(* Logix 5000 project; controller CarbonScout_MK6 vendor 1 type 14 code 154 rev 32.11; software revision 32.00 *)
// CarbonScout_MK6

TASK DataMapping (periodic, rate 200 ms, priority 15, watchdog 1000 ms) : DataMapping
TASK Instruments (periodic, rate 100 ms, priority 8, watchdog 3000 ms) : Analogs, Valves
TASK Sequence (periodic, rate 150 ms, priority 12, watchdog 3000 ms) : SeqProgram
TASK System (periodic, rate 100 ms, priority 15, watchdog 2000 ms) : SystemTask

MODULES
   Local : vendor 1 type 14 code 154 (PointIO 0, rev 32.11)
      N206_pH_DO : vendor 1182 type 43 code 4252 (Ethernet 192.168.50.206, rev 2.1, Output RPI 100 ms)
      N205_Val : vendor 87 type 8640 code 8640 (Ethernet 192.168.50.205, rev 1.1, StandardDataDriven RPI 100 ms)
      Local02 : vendor 1 type 115 code 210 (PointIO 2, rev 3.1, Input RPI 100 ms)
           Local:2:I.Ch0Data   // LIT01 Laser
           Local:2:I.Ch4Data   // WIT01 Weightometer
           Local:2:I.Ch6Data   // Discharge Level
           Local:2:I.Ch5Data   // Booster Level
           Local:2:I.Ch1Data   // LIT02 Cone Level
           Local:2:I.Ch3Data   // PIT01 Water Flow
           Local:2:I.Ch2Data   // FIT01 Water Flow
      Discrete_IO : Embedded (PointIO 1, rev 32.11, Output RPI 20 ms)
           Local:1:I.Data.4   // Booster Contactor Closed
           Local:1:I.Data.7   // Discharge Contactor Closed
           Local:1:I.Data.3   // Booster CB healthy
           Local:1:I.Data.5   // Booster OL Tripped
           Local:1:I.Data.1   // XRF door switch
           Local:1:I.Data.2   // XRF Door Closed
           Local:1:I.Data.6   // Discharge CB Healthy
           Local:1:I.Data.0   // Low Air Pressure
           Local:1:I.Data.8   // Discharge OL Tripped
           Local:1:O.Data.10   // XV36
           Local:1:O.Data.5   // XV31
           Local:1:O.Data.6   // XV32
           Local:1:O.Data.7   // XV33
           Local:1:O.Data.14   // Discharge Pump Stop
           Local:1:O.Data.0   // Green
           Local:1:O.Data.1   // Amber
           Local:1:O.Data.3   // PC Relay
           Local:1:O.Data.8   // XV34
           Local:1:O.Data.9   // XV35
           Local:1:O.Data.4   // XRF Relay
           Local:1:O.Data.12   // Booster Pump Stop
           Local:1:O.Data.2   // Red
           Local:1:O.Data.11   // Booster Pump Start
           Local:1:O.Data.13   // Discharge pump Start
END_MODULES

TYPE CS_Results :
STRUCT
   Run_ID : DINT;   // RunID
   Carbon_VOL_ml : REAL;   // Carbon Volume
   Carbon_MASS : REAL;   // Calculated Carbon Weight (g)
   Carbon_DIST : REAL;   // Calcaulted Carbon Distribution g/L
   Hour : DINT;   // Sample Hour
   Min : DINT;   // Sample Minute
   Day : DINT;   // Sample Day
   Month : DINT;   // Sample Month
   Year : DINT;   // Sample Year
   Sample_DO : REAL;   // Measured DO
   Sample_pH : REAL;   // Measured pH
   Sample_VOL : REAL;   // Measured Slurry Volume (L)
   Au : REAL;   // XRF
   CN : REAL;   // CN
   Density : REAL;   // % Solids
   EmptyDist : REAL;   // Laser Empty Measurement (mm)
   FullDist : REAL;   // Laser Carbon Level Measurement (mm)
   ErrorFlag : DINT;   // Sample Error Flag
   Carbon_mLperL : REAL;   // Carbon mL/L
   Slurry_Weight : REAL;   // Measured Slurry Weight (Kg)
   Sample_ORP : REAL;   // Measured ORP
   Sample_Temperature_pH : REAL;   // Measured Temperautre from pH probe
   Sample_Temperature_DO : REAL;   // Measured Temperautre from DO probe
   Sample_Tank : DINT;   // Tank Index Tank1=1 Tank 2 = 2 ect
   Carbon_Height : REAL;   // EmptyDistance - Full Distance (mm)
   Sample_FlowRate : REAL;   // Sample Flow Rate L/s
   Sample_FillTime : REAL;   // Solution Feel Time
   PurgeWaterUsed : REAL;   // Purge Water Used
   DisplacedCarbonVol : REAL;   // Displaced carbon volume
   DisplacedCarbonMass : REAL;   // Displaced carbon Mass
   SampleDuration : DINT;   // Sec
END_STRUCT
END_TYPE

TYPE CS_TankParams :
STRUCT
   Run_ID : DINT;
   Sample_Cnt : DINT;
   Sample_Time : DINT;
   NoFill_TimeOut : DINT;
   Purge_Time : DINT;
   Online : BOOL;
   LogTrigger : BOOL;
   Name : STRING_20;
   CarbonSP : REAL;
   From : DINT;
   To : DINT;
   XferPump : BOOL;
   PumpRunTime : REAL;   // Minutes
   Volume : REAL;   // CIL/CIP tank capacity (ton)
   LineBlock : BOOL;
   LineBreak : BOOL;
   PurgeLow : BOOL;
   TotalCarbonMass : REAL;   // kg
   GoldMass : REAL;   // kg
   LiquidDensity : REAL;   // SG
   SolidsDensity : REAL;   // SG
   LeachOnly : BOOL;   // 1= Leach Only, Carbon measurement&XRF skip 0= Adsoption
   PurgeVolume : REAL;   // Purge Volume
END_STRUCT
END_TYPE

TYPE GEK_Sequence :
STRUCT
   Mode : P_Mode;
   POC : GekkoSeq;
   ActiveStage : DINT;
   SeqTimer : TIMER[2];
   HMI_Start_Req : BOOL;
   HMI_StopPause_Req : BOOL;
   HMI_Pause_Req : BOOL;
   HMI_SkipF_Req : BOOL;
   HMI_SkipR_Req : BOOL;
   HMI_Resume_Req : BOOL;
   Group_ProgRel_Req : BOOL;
   Group_ProgLock_Req : BOOL;
   Group_ProgUnLock_Req : BOOL;
   Group_ProgAcq_Req : BOOL;
   HMI_Stop_Req : BOOL;
   AlarmsFlags : DINT[1];
   HMI_Reset_Req : BOOL;
END_STRUCT
END_TYPE

TYPE LinearModel :
STRUCT
   A : REAL;   // Gradient Coefficient
   B : REAL;   // Intercept/Offset Constant
END_STRUCT
END_TYPE

TYPE LinearModelXRF :
STRUCT
   Au_Scaled : REAL;
   Au_ErrScaled : REAL;
   Au_Raw : REAL;
   Au_ErrRaw : REAL;
   Au_Model : LinearModel[2];
   Mg_Scaled : REAL;
   Mg_ErrScaled : REAL;
   Mg_Raw : REAL;
   Mg_ErrRaw : REAL;
   Mg_Model : LinearModel[2];
   Al_Scaled : REAL;
   Al_ErrScaled : REAL;
   Al_Raw : REAL;
   Al_ErrRaw : REAL;
   Al_Model : LinearModel[2];
   Si_Scaled : REAL;
   Si_ErrScaled : REAL;
   Si_Raw : REAL;
   Si_ErrRaw : REAL;
   Si_Model : LinearModel[2];
   P_Scaled : REAL;
   P_ErrScaled : REAL;
   P_Raw : REAL;
   P_ErrRaw : REAL;
   P_Model : LinearModel[2];
   S_Scaled : REAL;
   S_ErrScaled : REAL;
   S_Raw : REAL;
   S_ErrRaw : REAL;
   S_Model : LinearModel[2];
   K_Scaled : REAL;
   K_ErrScaled : REAL;
   K_Raw : REAL;
   K_ErrRaw : REAL;
   K_Model : LinearModel[2];
   Ca_Scaled : REAL;
   Ca_ErrScaled : REAL;
   Ca_Raw : REAL;
   Ca_ErrRaw : REAL;
   Ca_Model : LinearModel[2];
   Ti_Scaled : REAL;
   Ti_ErrScaled : REAL;
   Ti_Raw : REAL;
   Ti_ErrRaw : REAL;
   Ti_Model : LinearModel[2];
   V_Scaled : REAL;
   V_ErrScaled : REAL;
   V_Raw : REAL;
   V_ErrRaw : REAL;
   V_Model : LinearModel[2];
   Cr_Scaled : REAL;
   Cr_ErrScaled : REAL;
   Cr_Raw : REAL;
   Cr_ErrRaw : REAL;
   Cr_Model : LinearModel[2];
   Mn_Scaled : REAL;
   Mn_ErrScaled : REAL;
   Mn_Raw : REAL;
   Mn_ErrRaw : REAL;
   Mn_Model : LinearModel[2];
   Fe_Scaled : REAL;
   Fe_ErrScaled : REAL;
   Fe_Raw : REAL;
   Fe_ErrRaw : REAL;
   Fe_Model : LinearModel[2];
   Co_Scaled : REAL;
   Co_ErrScaled : REAL;
   Co_Raw : REAL;
   Co_ErrRaw : REAL;
   Co_Model : LinearModel[2];
   Ni_Scaled : REAL;
   Ni_ErrScaled : REAL;
   Ni_Raw : REAL;
   Ni_ErrRaw : REAL;
   Ni_Model : LinearModel[2];
   Cu_Scaled : REAL;
   Cu_ErrScaled : REAL;
   Cu_Raw : REAL;
   Cu_ErrRaw : REAL;
   Cu_Model : LinearModel[2];
   Zn_Scaled : REAL;
   Zn_ErrScaled : REAL;
   Zn_Raw : REAL;
   Zn_ErrRaw : REAL;
   Zn_Model : LinearModel[2];
   As_Scaled : REAL;
   As_ErrScaled : REAL;
   As_Raw : REAL;
   As_ErrRaw : REAL;
   As_Model : LinearModel[2];
   Se_Scaled : REAL;
   Se_ErrScaled : REAL;
   Se_Raw : REAL;
   Se_ErrRaw : REAL;
   Se_Model : LinearModel[2];
   Rb_Scaled : REAL;
   Rb_ErrScaled : REAL;
   Rb_Raw : REAL;
   Rb_ErrRaw : REAL;
   Rb_Model : LinearModel[2];
   Sr_Scaled : REAL;
   Sr_ErrScaled : REAL;
   Sr_Raw : REAL;
   Sr_ErrRaw : REAL;
   Sr_Model : LinearModel[2];
   Y_Scaled : REAL;
   Y_ErrScaled : REAL;
   Y_Raw : REAL;
   Y_ErrRaw : REAL;
   Y_Model : LinearModel[2];
   Zr_Scaled : REAL;
   Zr_ErrScaled : REAL;
   Zr_Raw : REAL;
   Zr_ErrRaw : REAL;
   Zr_Model : LinearModel[2];
   Nb_Scaled : REAL;
   Nb_ErrScaled : REAL;
   Nb_Raw : REAL;
   Nb_ErrRaw : REAL;
   Nb_Model : LinearModel[2];
   Mo_Scaled : REAL;
   Mo_ErrScaled : REAL;
   Mo_Raw : REAL;
   Mo_ErrRaw : REAL;
   Mo_Model : LinearModel[2];
   Ag_Scaled : REAL;
   Ag_ErrScaled : REAL;
   Ag_Raw : REAL;
   Ag_ErrRaw : REAL;
   Ag_Model : LinearModel[2];
   Cd_Scaled : REAL;
   Cd_ErrScaled : REAL;
   Cd_Raw : REAL;
   Cd_ErrRaw : REAL;
   Cd_Model : LinearModel[2];
   Sn_Scaled : REAL;
   Sn_ErrScaled : REAL;
   Sn_Raw : REAL;
   Sn_ErrRaw : REAL;
   Sn_Model : LinearModel[2];
   Sb_Scaled : REAL;
   Sb_ErrScaled : REAL;
   Sb_Raw : REAL;
   Sb_ErrRaw : REAL;
   Sb_Model : LinearModel[2];
   Ba_Scaled : REAL;
   Ba_ErrScaled : REAL;
   Ba_Raw : REAL;
   Ba_ErrRaw : REAL;
   Ba_Model : LinearModel[2];
   La_Scaled : REAL;
   La_ErrScaled : REAL;
   La_Raw : REAL;
   La_ErrRaw : REAL;
   La_Model : LinearModel[2];
   Ce_Scaled : REAL;
   Ce_ErrScaled : REAL;
   Ce_Raw : REAL;
   Ce_ErrRaw : REAL;
   Ce_Model : LinearModel[2];
   Pr_Scaled : REAL;
   Pr_ErrScaled : REAL;
   Pr_Raw : REAL;
   Pr_ErrRaw : REAL;
   Pr_Model : LinearModel[2];
   Nd_Scaled : REAL;
   Nd_ErrScaled : REAL;
   Nd_Raw : REAL;
   Nd_ErrRaw : REAL;
   Nd_Model : LinearModel[2];
   W_Scaled : REAL;
   W_ErrScaled : REAL;
   W_Raw : REAL;
   W_ErrRaw : REAL;
   W_Model : LinearModel[2];
   Hg_Scaled : REAL;
   Hg_ErrScaled : REAL;
   Hg_Raw : REAL;
   Hg_ErrRaw : REAL;
   Hg_Model : LinearModel[2];
   Pb_Scaled : REAL;
   Pb_ErrScaled : REAL;
   Pb_Raw : REAL;
   Pb_ErrRaw : REAL;
   Pb_Model : LinearModel[2];
   Bi_Scaled : REAL;
   Bi_ErrScaled : REAL;
   Bi_Raw : REAL;
   Bi_ErrRaw : REAL;
   Bi_Model : LinearModel[2];
   Th_Scaled : REAL;
   Th_ErrScaled : REAL;
   Th_Raw : REAL;
   Th_ErrRaw : REAL;
   Th_Model : LinearModel[2];
   U_Scaled : REAL;
   U_ErrScaled : REAL;
   U_Raw : REAL;
   U_ErrRaw : REAL;
   U_Model : LinearModel[2];
   LE_Scaled : REAL;
   LE_ErrScaled : REAL;
   LE_Raw : REAL;
   LE_ErrRaw : REAL;
   LE_Model : LinearModel[2];
   Default : BOOL;
   Save : BOOL;
   Restore : BOOL;
END_STRUCT
END_TYPE

TYPE STRING_12 :
STRUCT
   LEN : DINT;
   DATA : SINT[12];
END_STRUCT
END_TYPE

TYPE STRING_16 :
STRUCT
   LEN : DINT;
   DATA : SINT[16];
END_STRUCT
END_TYPE

TYPE STRING_20 :
STRUCT
   LEN : DINT;
   DATA : SINT[20];
END_STRUCT
END_TYPE

TYPE String_30 :
STRUCT
   LEN : DINT;
   DATA : SINT[30];
END_STRUCT
END_TYPE

TYPE String_4 :
STRUCT
   LEN : DINT;
   DATA : SINT[4];
END_STRUCT
END_TYPE

TYPE STRING_40 :
STRUCT
   LEN : DINT;
   DATA : SINT[40];
END_STRUCT
END_TYPE

TYPE STRING_8 :
STRUCT
   LEN : DINT;
   DATA : SINT[8];
END_STRUCT
END_TYPE

TYPE XRF :   // XRF data
STRUCT
   Run_ID : DINT;
   OCmd_Start : BOOL;
   OCmd_Stop : BOOL;
   Out_Run : BOOL;
   PCmd_Run : BOOL;
   Sts_Ready : BOOL;
   Sts_CommLoss : BOOL;
   ModbusDINT_IN : DINT[3];
   ModbusINT_OUT : DINT[20];
   ModbusBOOL_IN : BOOL[32];
   ModbusBOOL_OUT : BOOL[32];
   Results : DINT[150];
   Mode : BOOL;   // 0 = Manual, 1 = Auto
   OCmd_SetBeam : BOOL;
   Sts_Running : BOOL;
   Sts_Fault : BOOL;
   Sts_Powered : BOOL;
   Sts_Intlk : BOOL;
   Sts_Perm : BOOL;
   Inp_Sim : BOOL;
   Modes : P_Mode;
   Sts_WarmUp : BOOL;
   Sts_LastBootTime : INT;   // Seconds to ready from power on
END_STRUCT
END_TYPE

ADD_ON_INSTRUCTION GekkoSeq   (* revision 1.3 *)
// Revision note:
// V1.0 - Barry T Idea
// V1.1 - Travis L implemented
// V1.2 - Minor Bug Fixes ( Resumed too quick, it doesnt have any status)
// V1.3 - Minor Bug Fixes (Stop Paused and Paused at the same time unlatch Sts_Paused
// V1.3 - Intlk01 and Intlk02 added for Pause intlk and stop Pause intlk. Cfg_Intlk is removed
// Help:
// Intented Purpose
// In_Cfg_BatchContinous - Set to batch x= 1 for equipment that has descrete stages that can be switched between Eg. ILR
// In_Cfg_BatchContinous - Set to continous x=0 for equipment where the sequence should return to idle if paused/stopped.
// In_IntlkOk1 = 0 Stop pause will be initiated on interlock trip/Control Stop will be initiated on sequence.
// In_IntlkOK2 = 0 Pause will be initiated on interlock trip.
// Pause command will stop the sequence at the current step and retain the step timer. Resuming will contrinue exactly where paused.
// StopPuase command will stop the sequence at the current step and reset the step timer. Resuming will start the current selected step from the start.
VAR_INPUT
   In_Cfg_BatchContinous : BOOL; {visible}   // Configuration - 0 = Continuous 1= Batch
   In_Cmd_Start : BOOL; {visible}   // 1= Request start
   In_PermOK : BOOL; {visible}   // 1= Permissives to start are OK
   In_Intlk1OK : BOOL; {visible}   // 1= Stop Pause Interlocks are ok / Control Stop on Continuous
   In_Cmd_Stop : BOOL; {visible}   // 1= Command a controlled sequence stop
END_VAR
VAR_OUTPUT
   Out_Run : BOOL; {visible}   // 1= Sequence block in Run state
END_VAR
VAR_INPUT
   In_Running : BOOL; {visible}   // 1= Running feedback from sequence
END_VAR
VAR_OUTPUT
   Sts_Running : BOOL; {access Read Only, visible}   // 1= Sequence is running
   Sts_Starting : BOOL; {access Read Only, visible}   // 1= Sequence is starting (waiting for running feedback)
   Sts_Stopped : BOOL; {access Read Only, visible}   // 1= Sequence is stopped and in Idle State
   Sts_Stopping : BOOL; {access Read Only, visible}   // 1= Sequence is stopping (waiting for stopped feedback)
END_VAR
VAR_INPUT
   In_Stopped : BOOL; {visible}   // 1= Stopped feedback from sequence (Sequence is Idle)
   In_Cmd_StopPause : BOOL; {visible}   // 1= Command a StopPause of the sequence (Pauses sequence and reset timers)
   In_Cmd_Pause : BOOL; {visible}   // 1= Command Pauses sequence. Retains step timers
   In_Cmd_Resume : BOOL; {visible}   // 1= Command Resume of sequence
END_VAR
VAR_OUTPUT
   Sts_StopPaused : BOOL; {access Read Only, visible}   // 1= Sequence is StopPaused. Timers Reset
   Sts_Paused : BOOL; {access Read Only, visible}   // 1= Sequence is paused. Timers Retained
END_VAR
VAR_IN_OUT
   Out_StepTm : TIMER; {required}   // Accumulated Step Time (sec)
END_VAR
VAR_INPUT
   In_StepNum : DINT; {visible}   // Requested step number
END_VAR
VAR_OUTPUT
   Out_NewStepNum : DINT; {access Read Only, visible}   // Step number that will be run upon sequence running
   Sts_Skipped : BOOL; {access Read Only, visible}   // 1= Sequence step has been skipped
END_VAR
VAR_INPUT
   In_Cmd_SkipF : BOOL; {visible}   // 1= Command sequence to skip foward one step number
   In_Cmd_SkipR : BOOL; {visible}   // 1= Command sequence to skip backwards one step number
   In_MaxStepNum : DINT; {visible}   // Maximum step number of sequence
END_VAR
VAR_OUTPUT
   Sts_Resumed : BOOL; {access Read Only, visible}   // Resumed Oneshot
   Sts_OKToStart : BOOL; {access Read Only, visible}
   Out_MovingStepNum : DINT; {access Read Only, visible}
END_VAR
VAR_INPUT
   In_Intlk2OK : BOOL;   // 1= Pause Interlocks are ok
END_VAR
VAR
   Local_RunningDB : TIMER := (PRE := 100); {access None}
   Local_Oneshot : DINT; {access None}
   Local_MovingStepNum : DINT; {access None}
   Local_StepTm_Stored : DINT; {access None}
END_VAR

ROUTINE Logic   (* ladder *)
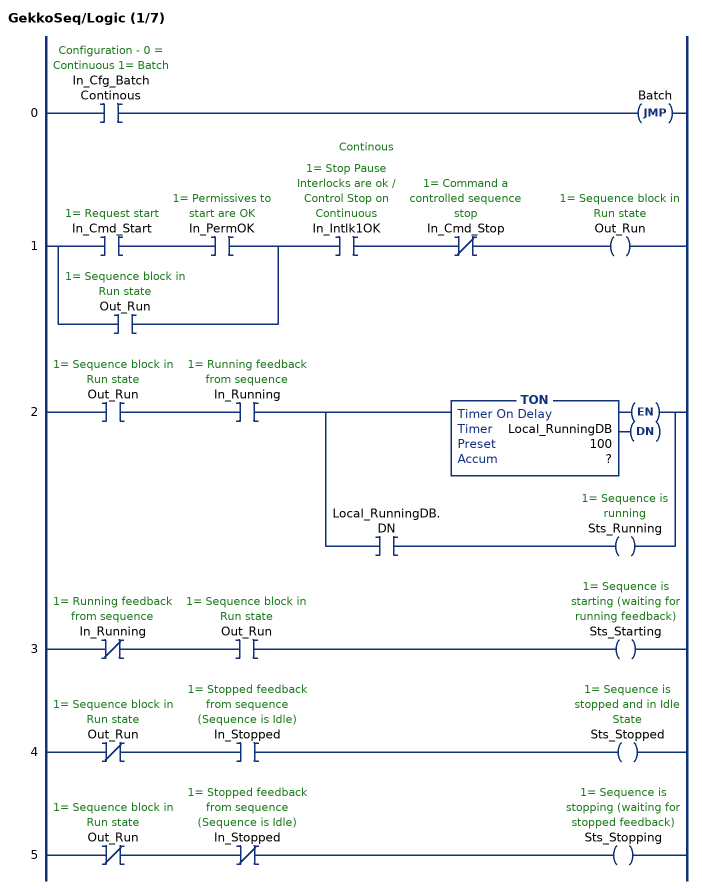
   0: XIC(In_Cfg_BatchContinous)JMP(Batch);
   // Continous
   1: [XIC(In_Cmd_Start) XIC(In_PermOK) ,XIC(Out_Run) ]XIC(In_Intlk1OK)XIO(In_Cmd_Stop)OTE(Out_Run);
   2: XIC(Out_Run)XIC(In_Running)[TON(Local_RunningDB,?,?) ,XIC(Local_RunningDB.DN) OTE(Sts_Running) ];
   3: XIO(In_Running)XIC(Out_Run)OTE(Sts_Starting);
   4: XIO(Out_Run)XIC(In_Stopped)OTE(Sts_Stopped);
   5: XIO(Out_Run)XIO(In_Stopped)OTE(Sts_Stopping);
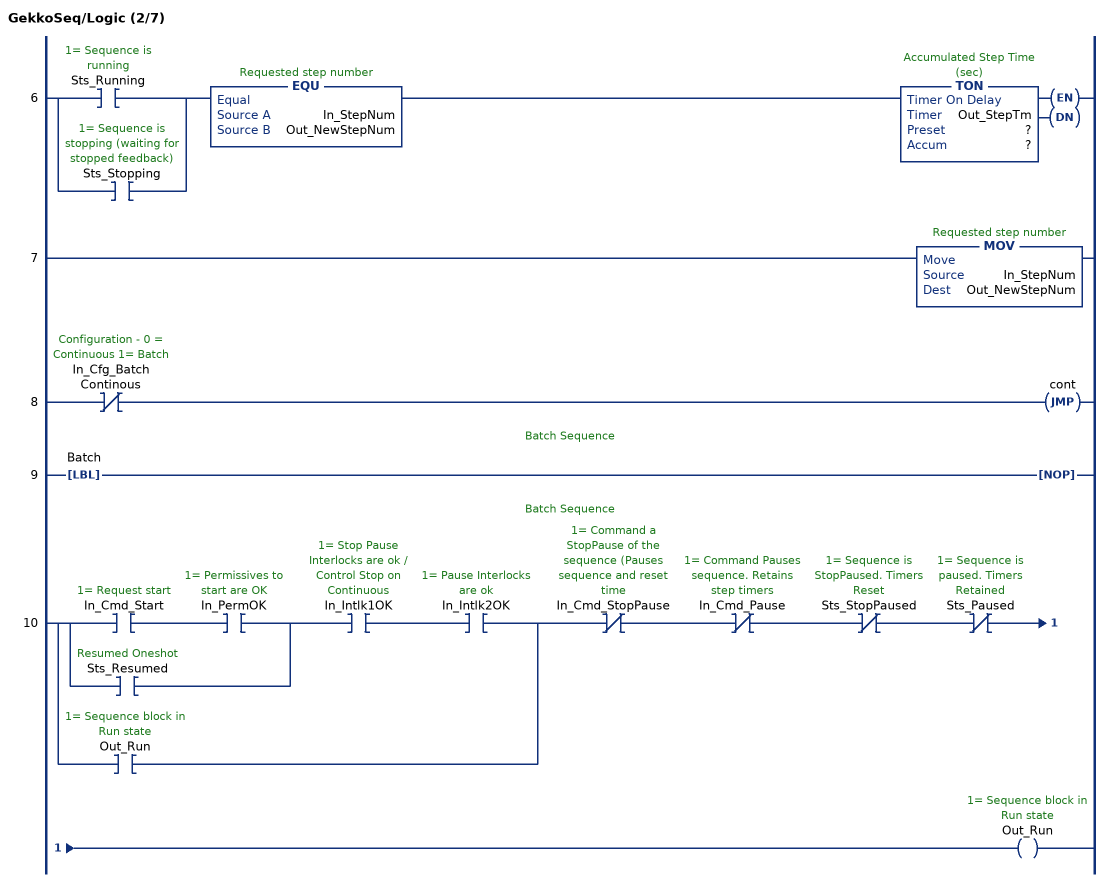
   6: [XIC(Sts_Running) ,XIC(Sts_Stopping) ]EQU(In_StepNum,Out_NewStepNum)TON(Out_StepTm,?,?);
   7: MOV(In_StepNum,Out_NewStepNum);
   8: XIO(In_Cfg_BatchContinous)JMP(cont);
   // Batch Sequence
   9: LBL(Batch)NOP();
   // Batch Sequence
   10: [[XIC(In_Cmd_Start) XIC(In_PermOK) ,XIC(Sts_Resumed) ] XIC(In_Intlk1OK) XIC(In_Intlk2OK) ,XIC(Out_Run) ]XIO(In_Cmd_StopPause)XIO(In_Cmd_Pause)XIO(Sts_StopPaused)XIO(Sts_Paused)OTE(Out_Run);
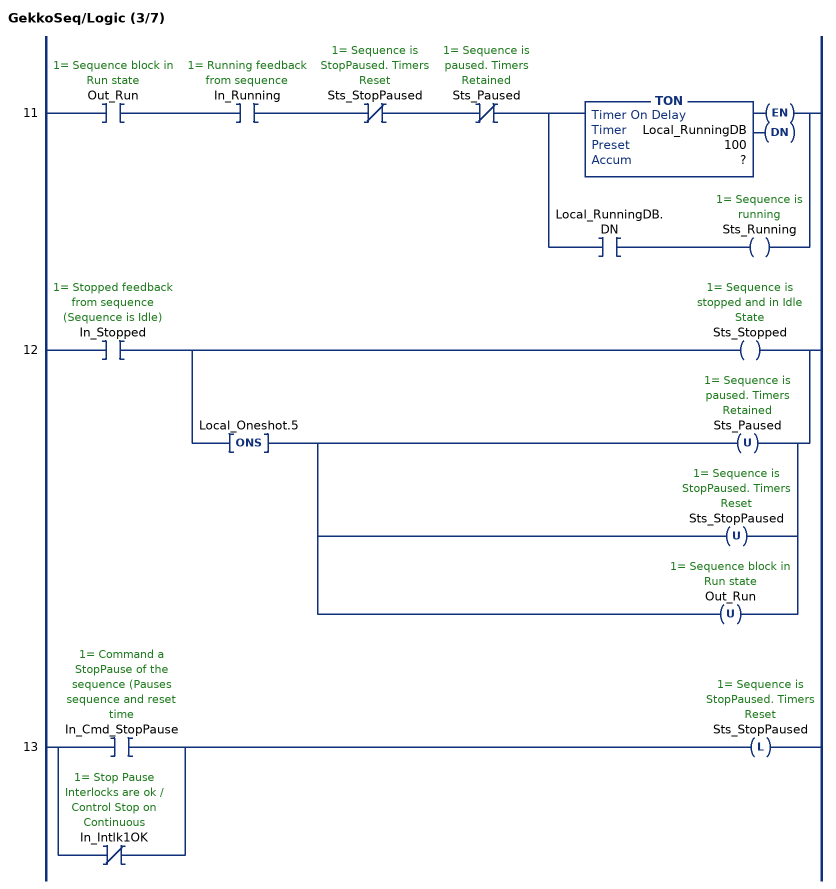
   11: XIC(Out_Run)XIC(In_Running)XIO(Sts_StopPaused)XIO(Sts_Paused)[TON(Local_RunningDB,?,?) ,XIC(Local_RunningDB.DN) OTE(Sts_Running) ];
   12: XIC(In_Stopped)[OTE(Sts_Stopped) ,ONS(Local_Oneshot.5) [OTU(Sts_Paused) ,OTU(Sts_StopPaused) ,OTU(Out_Run) ] ];
   13: [XIC(In_Cmd_StopPause) ,XIO(In_Intlk1OK) ]OTL(Sts_StopPaused);
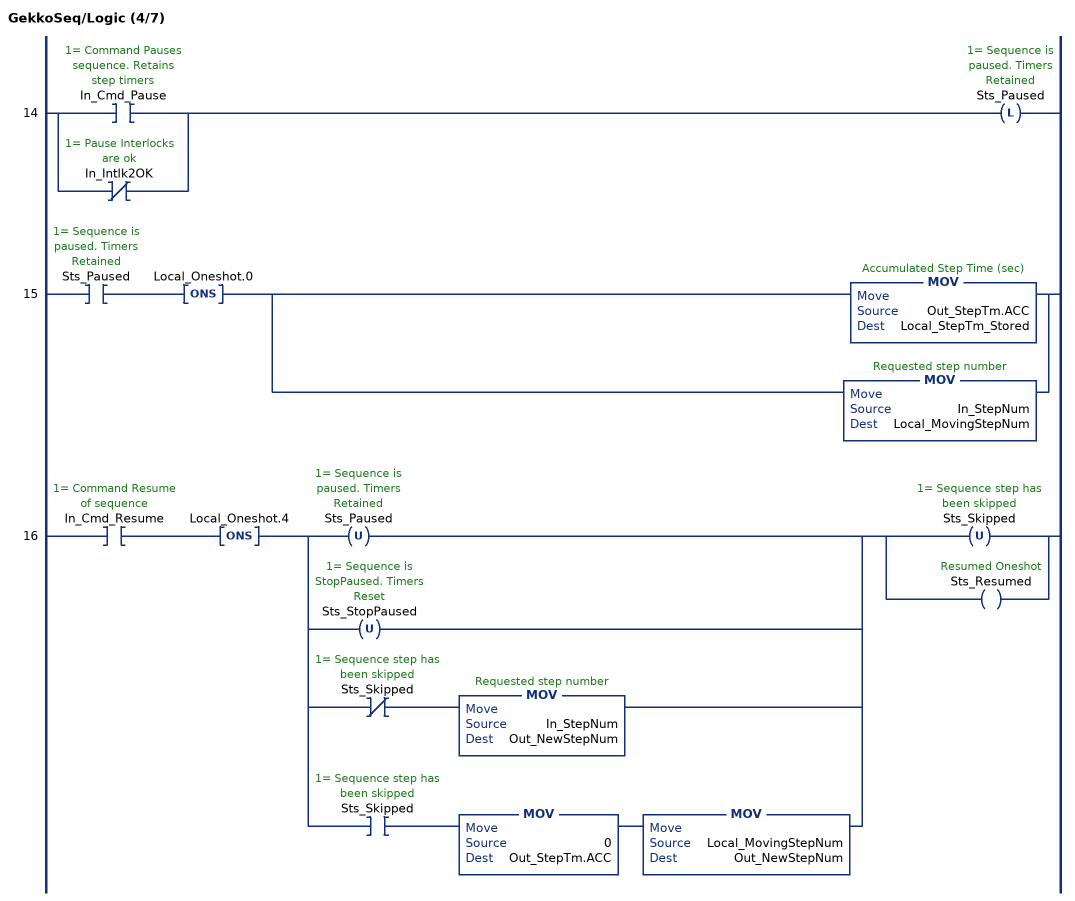
   14: [XIC(In_Cmd_Pause) ,XIO(In_Intlk2OK) ]OTL(Sts_Paused);
   15: XIC(Sts_Paused)ONS(Local_Oneshot.0)[MOV(Out_StepTm.ACC,Local_StepTm_Stored) ,MOV(In_StepNum,Local_MovingStepNum) ];
   16: XIC(In_Cmd_Resume)ONS(Local_Oneshot.4)[OTU(Sts_Paused) ,OTU(Sts_StopPaused) ,XIO(Sts_Skipped) MOV(In_StepNum,Out_NewStepNum) ,XIC(Sts_Skipped) MOV(0,Out_StepTm.ACC) MOV(Local_MovingStepNum,Out_NewStepNum) ][OTU(Sts_Skipped) ,OTE(Sts_Resumed) ];
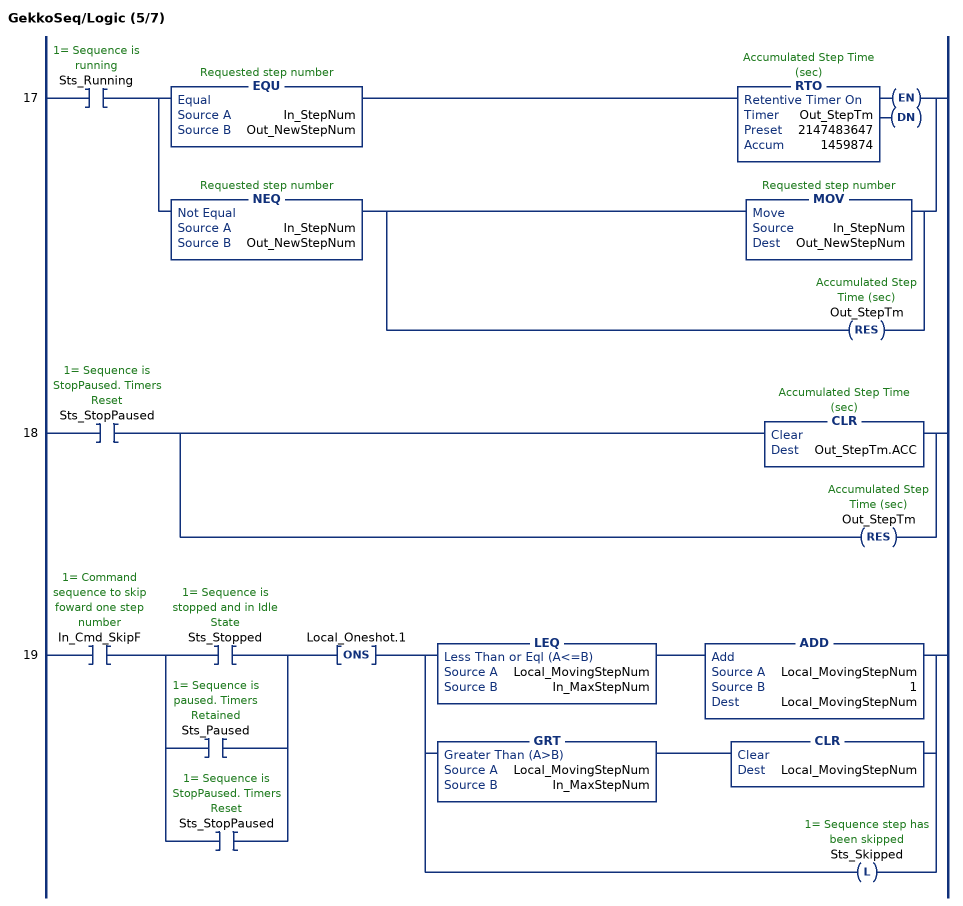
   17: XIC(Sts_Running)[EQU(In_StepNum,Out_NewStepNum) RTO(Out_StepTm,2147483647,1459874) ,NEQ(In_StepNum,Out_NewStepNum) [MOV(In_StepNum,Out_NewStepNum) ,RES(Out_StepTm) ] ];
   18: XIC(Sts_StopPaused)[CLR(Out_StepTm.ACC) ,RES(Out_StepTm) ];
   19: XIC(In_Cmd_SkipF)[XIC(Sts_Stopped) ,XIC(Sts_Paused) ,XIC(Sts_StopPaused) ]ONS(Local_Oneshot.1)[LEQ(Local_MovingStepNum,In_MaxStepNum) ADD(Local_MovingStepNum,1,Local_MovingStepNum) ,GRT(Local_MovingStepNum,In_MaxStepNum) CLR(Local_MovingStepNum) ,OTL(Sts_Skipped) ];
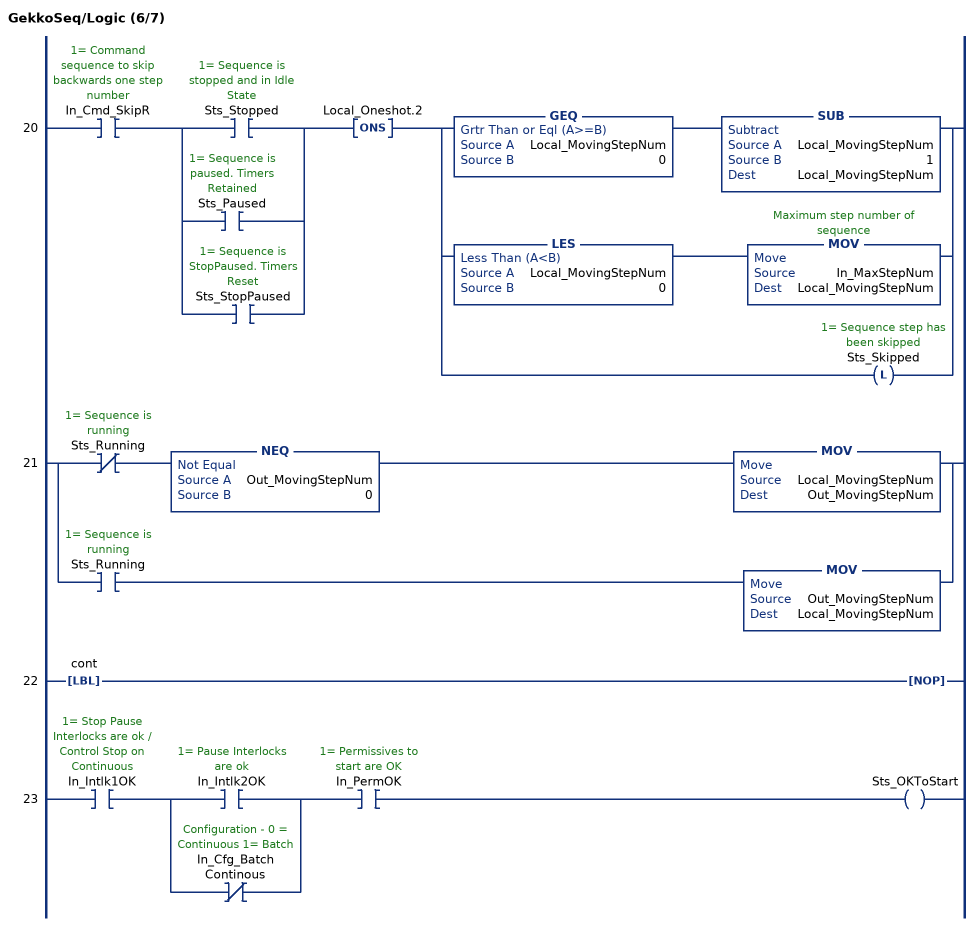
   20: XIC(In_Cmd_SkipR)[XIC(Sts_Stopped) ,XIC(Sts_Paused) ,XIC(Sts_StopPaused) ]ONS(Local_Oneshot.2)[GEQ(Local_MovingStepNum,0) SUB(Local_MovingStepNum,1,Local_MovingStepNum) ,LES(Local_MovingStepNum,0) MOV(In_MaxStepNum,Local_MovingStepNum) ,OTL(Sts_Skipped) ];
   21: [XIO(Sts_Running) NEQ(Out_MovingStepNum,0) MOV(Local_MovingStepNum,Out_MovingStepNum) ,XIC(Sts_Running) MOV(Out_MovingStepNum,Local_MovingStepNum) ];
   22: LBL(cont)NOP();
   23: XIC(In_Intlk1OK)[XIC(In_Intlk2OK) ,XIO(In_Cfg_BatchContinous) ]XIC(In_PermOK)OTE(Sts_OKToStart);
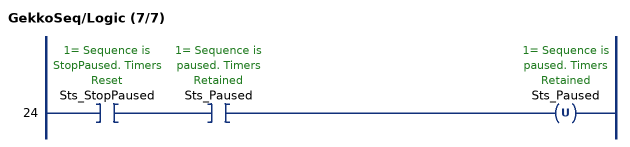
   24: XIC(Sts_StopPaused)XIC(Sts_Paused)OTU(Sts_Paused);
END_ROUTINE
END_ADD_ON_INSTRUCTION

ADD_ON_INSTRUCTION GekkoValvePulse   (* revision 1.0, ExecutePrescan *)
VAR_INPUT
   OnTime : DINT; {required}
   OffTime : DINT; {required}
END_VAR
VAR_OUTPUT
   Out_Open : BOOL; {access Read Only}
END_VAR
VAR
   OnTimer : TIMER; {access None}
   OffTimer : TIMER; {access None}
END_VAR

ROUTINE Logic   (* ladder *)
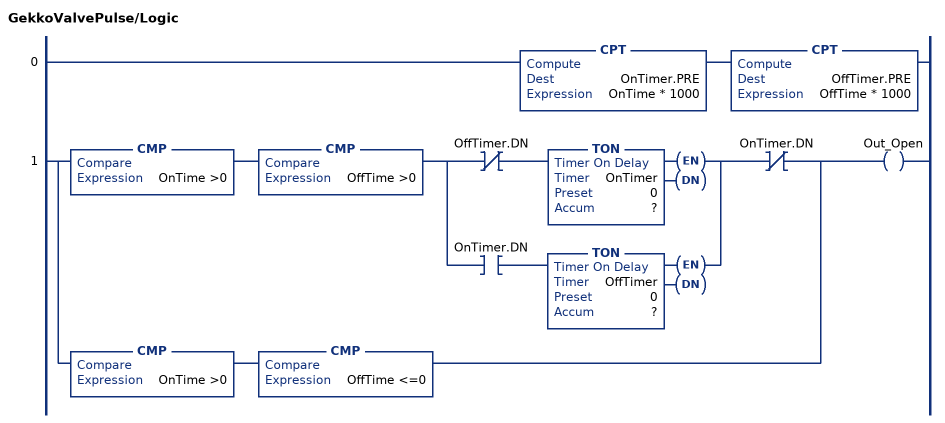
   0: CPT(OnTimer.PRE,OnTime * 1000)CPT(OffTimer.PRE,OffTime * 1000);
   1: [CMP(OnTime >0) CMP(OffTime >0) [XIO(OffTimer.DN) TON(OnTimer,?,?) ,XIC(OnTimer.DN) TON(OffTimer,?,?) ] XIO(OnTimer.DN) ,CMP(OnTime >0) CMP(OffTime <=0) ]OTE(Out_Open);
END_ROUTINE

ROUTINE Prescan   (* ladder *)
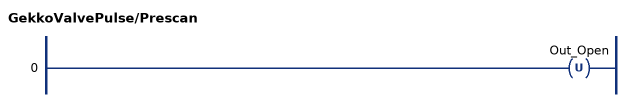
   0: OTU(Out_Open);
END_ROUTINE
END_ADD_ON_INSTRUCTION

ADD_ON_INSTRUCTION GekkoValveStat   (* revision 1.0 *)
VAR_INPUT
   Inp_Opened : BOOL; {required}
   Inp_Closed : BOOL; {required}
END_VAR
VAR_OUTPUT
   Out_OpenCNT : REAL; {visible}
   Out_CloseCNT : REAL; {visible}
END_VAR
VAR_INPUT
   Inp_OpenCNTReset : BOOL; {visible}
   Inp_CloseCNTReset : BOOL; {visible}
   Inp_OpenCNTSP : REAL;
   Inp_CloseCNTSP : REAL;
END_VAR
VAR_OUTPUT
   Out_OpenReached : BOOL; {access Read Only}
   Out_CloseReached : BOOL; {access Read Only}
END_VAR
VAR
   WrkONS : BOOL[32]; {access None}
END_VAR

ROUTINE Logic   (* ladder *)
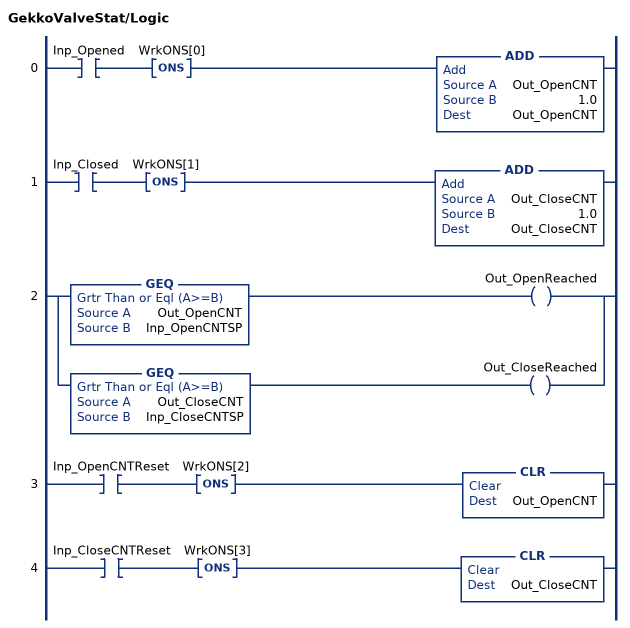
   0: XIC(Inp_Opened)ONS(WrkONS[0])ADD(Out_OpenCNT,1.0,Out_OpenCNT);
   1: XIC(Inp_Closed)ONS(WrkONS[1])ADD(Out_CloseCNT,1.0,Out_CloseCNT);
   2: [GEQ(Out_OpenCNT,Inp_OpenCNTSP) OTE(Out_OpenReached) ,GEQ(Out_CloseCNT,Inp_CloseCNTSP) OTE(Out_CloseReached) ];
   3: XIC(Inp_OpenCNTReset)ONS(WrkONS[2])CLR(Out_OpenCNT);
   4: XIC(Inp_CloseCNTReset)ONS(WrkONS[3])CLR(Out_CloseCNT);
END_ROUTINE
END_ADD_ON_INSTRUCTION

ADD_ON_INSTRUCTION LookUpTable   (* revision 1.2, vendor Rockwell Automation *)
// Look Up Table
// Help:
// Use this instruction to scale data from your analog module and bring it into the limits prescribed by the process variable or another analog module.
// Equations used in calculating a linear relationship:
// Scaled value = (input value - input min.) x rate + scaled minimum
// Rate = (scaled max. - scaled min.) / (input max. - input min.)
VAR_INPUT
   Input : REAL; {required}
   Y0 : REAL; {required}
   X1 : REAL; {required}
   Y1 : REAL; {required}
   X2 : REAL; {required}
   Y2 : REAL; {required}
   X3 : REAL; {required}
   Y3 : REAL; {required}
   X4 : REAL; {required}
   Y4 : REAL; {required}
   X5 : REAL; {required}
   Y5 : REAL; {required}
   X6 : REAL; {required}
   Y6 : REAL; {required}
   X7 : REAL; {required}
   Y7 : REAL; {required}
   X8 : REAL; {required}
   Y8 : REAL; {required}
   X9 : REAL; {required}
   Y9 : REAL; {required}
   X10 : REAL; {required}
   Y10 : REAL; {required}
END_VAR
VAR_OUTPUT
   Output : REAL; {access Read Only, required}
END_VAR
VAR
   Rate : REAL;
END_VAR

ROUTINE Logic   (* ladder *)
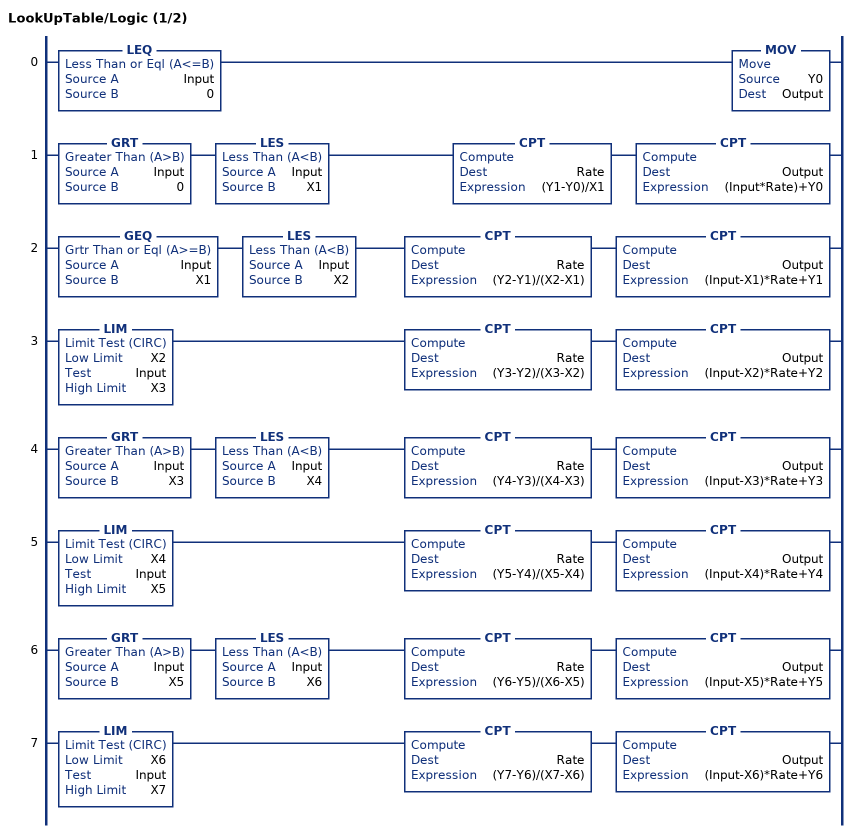
   0: LEQ(Input,0)MOV(Y0,Output);
   1: GRT(Input,0)LES(Input,X1)CPT(Rate,(Y1-Y0)/X1)CPT(Output,(Input*Rate)+Y0);
   2: GEQ(Input,X1)LES(Input,X2)CPT(Rate,(Y2-Y1)/(X2-X1))CPT(Output,(Input-X1)*Rate+Y1);
   3: LIM(X2,Input,X3)CPT(Rate,(Y3-Y2)/(X3-X2))CPT(Output,(Input-X2)*Rate+Y2);
   4: GRT(Input,X3)LES(Input,X4)CPT(Rate,(Y4-Y3)/(X4-X3))CPT(Output,(Input-X3)*Rate+Y3);
   5: LIM(X4,Input,X5)CPT(Rate,(Y5-Y4)/(X5-X4))CPT(Output,(Input-X4)*Rate+Y4);
   6: GRT(Input,X5)LES(Input,X6)CPT(Rate,(Y6-Y5)/(X6-X5))CPT(Output,(Input-X5)*Rate+Y5);
   7: LIM(X6,Input,X7)CPT(Rate,(Y7-Y6)/(X7-X6))CPT(Output,(Input-X6)*Rate+Y6);
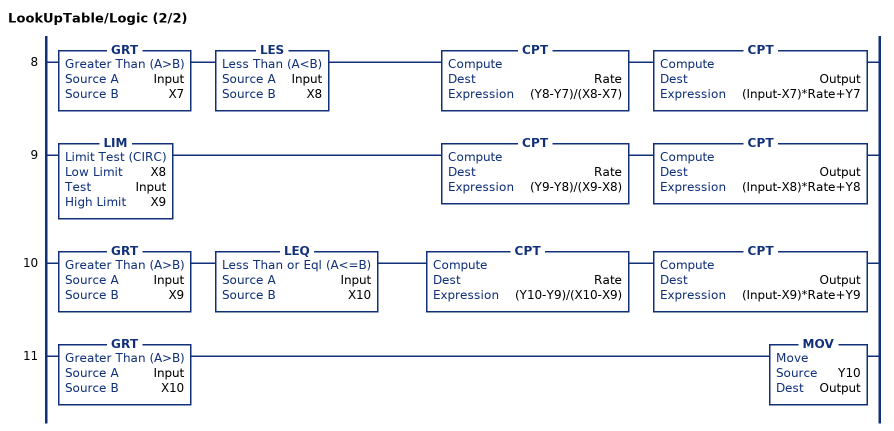
   8: GRT(Input,X7)LES(Input,X8)CPT(Rate,(Y8-Y7)/(X8-X7))CPT(Output,(Input-X7)*Rate+Y7);
   9: LIM(X8,Input,X9)CPT(Rate,(Y9-Y8)/(X9-X8))CPT(Output,(Input-X8)*Rate+Y8);
   10: GRT(Input,X9)LEQ(Input,X10)CPT(Rate,(Y10-Y9)/(X10-X9))CPT(Output,(Input-X9)*Rate+Y9);
   11: GRT(Input,X10)MOV(Y10,Output);
END_ROUTINE
END_ADD_ON_INSTRUCTION

ADD_ON_INSTRUCTION P_AIn   (* revision 3.5 02 Release, vendor Rockwell Automation, ExecutePrescan, ExecuteEnableInFalse *)
// Analog Input
// Revision note:
// See V3.5-xx Release Notes for details. Added Cfg_UseChanSrcQ to make SrcQ use independent of Cfg_HasChanObj, which is for navigation only.
// Help:
// Copyright © Rockwell Automation, Inc.  All Rights Reserved.
// This Instruction monitors an Analog Input from a flow, level, pressure,
// temperature, or any other analog sensor, and provides:
// *  Scaling, from Input (Raw) to PV (Engineering) Units
// *  High-High, High, Low and Low-Low Status and Alarms, with Gate
// inputs and configurable on-delay, off-delay and gate delay times
// *  Monitoring of bad/uncertain PV status, floating point exceptions
// and out-of-range conditions, with PV Fail alarm
// *  Setting of a simulated input signal for process simulation
// *  Capturing of the lowest and highest PV excursion values
// *  Program and Operator Settings for Status Thresholds
// *  Configurable threshold deadbands and out of range limits
// *  Maintenance Commands to allow manual override of the input signal (Substitute PV)
// Modes are provided by a P_Mode AOI instance.
// Alarms are provided by P_Alarm AOI instances.
// Status gating provided by P_Gate AOI instances.
// Modes of operation: Operator, Program, Maintenance
VAR_INPUT
   Inp_PV : REAL; {visible}   // Input Signal (process variable) from Sensor
   Inp_PVSrcQ : DINT;   // Input Source and Quality (from Channel object, if available) (enum)
   Inp_PVBad : BOOL; {visible}   // 1=PV or I/O Comms Status Bad, 0=OK
   Inp_PVUncertain : BOOL;   // 1=PV Value Not Reliable, 0=OK
   Inp_Sim : BOOL;   // 1=Use simulated PV (Set_SimPV); 0=Use Input (Inp_PV)
   Inp_HiHiGate : ALIAS FOR HiHiGate.Inp_Gate;   // High-High Status Gate, 1=enabled
   Inp_HiGate : ALIAS FOR HiGate.Inp_Gate;   // High Status Gate, 1=enabled
   Inp_LoGate : ALIAS FOR LoGate.Inp_Gate;   // Low Status Gate, 1=enabled
   Inp_LoLoGate : ALIAS FOR LoLoGate.Inp_Gate;   // Low-Low Status Gate, 1=enabled
   Inp_FailGate : ALIAS FOR FailGate.Inp_Gate;   // Fail Status Gate, 1=enabled
   Inp_Reset : BOOL; {visible}   // 1=Reset all Alarms requiring reset
   Cfg_NoSubstPV : BOOL;   // 1=Disallow selection of Substitute PV
   Cfg_SetTrack : BOOL := 1;   // 1=PSets track OSets in Oper, OSets track PSets in Prog, 0=no tracking
   Cfg_HasChanObj : BOOL;   // 1=Tells HMI a Channel object (AIChan, etc.) is used for Inp_PV
   Cfg_UseChanSrcQ : BOOL;   // 1=Pass thru connected Channel's SrcQ value, 0=generate SrcQ
   Cfg_PCmdClear : ALIAS FOR Mode.Cfg_PCmdClear;
   Cfg_ProgDefault : ALIAS FOR Mode.Cfg_ProgDefault;
   Cfg_HasHiHiAlm : ALIAS FOR HiHi.Cfg_Exists;   // 1=High-High Alarm exists and will be checked
   Cfg_HasHiAlm : ALIAS FOR Hi.Cfg_Exists;   // 1=High Alarm exists and will be checked
   Cfg_HasLoAlm : ALIAS FOR Lo.Cfg_Exists;   // 1=Low Alarm exists and will be checked
   Cfg_HasLoLoAlm : ALIAS FOR LoLo.Cfg_Exists;   // 1=Low-Low Alarm exists and will be checked
   Cfg_HasFailAlm : ALIAS FOR Fail.Cfg_Exists;   // 1=Analog Input Failure Alarm exists and will be checked
   Cfg_HiHiResetReqd : ALIAS FOR HiHi.Cfg_ResetReqd;   // 1=Reset required to clear High-High Alarm
   Cfg_HiResetReqd : ALIAS FOR Hi.Cfg_ResetReqd;   // 1=Reset required to clear High Alarm
   Cfg_LoResetReqd : ALIAS FOR Lo.Cfg_ResetReqd;   // 1=Reset required to clear Low Alarm
   Cfg_LoLoResetReqd : ALIAS FOR LoLo.Cfg_ResetReqd;   // 1=Reset required to clear Low-Low Alarm
   Cfg_FailResetReqd : ALIAS FOR Fail.Cfg_ResetReqd;   // 1=Reset required to clear Analog InputFailure Alarm
   Cfg_HiHiAckReqd : ALIAS FOR HiHi.Cfg_AckReqd;   // 1=Acknowledge required for High-High Alarm
   Cfg_HiAckReqd : ALIAS FOR Hi.Cfg_AckReqd;   // 1=Acknowledge required for High Alarm
   Cfg_LoAckReqd : ALIAS FOR Lo.Cfg_AckReqd;   // 1=Acknlowledge required for Low Alarm
   Cfg_LoLoAckReqd : ALIAS FOR LoLo.Cfg_AckReqd;   // 1=Acknowledge required for Low-Low Alarm
   Cfg_FailAckReqd : ALIAS FOR Fail.Cfg_AckReqd;   // 1=Acknowledge required for Analog Input Failure Alarm
   Cfg_HiHiSeverity : ALIAS FOR HiHi.Cfg_Severity;   // High-High Alarm Severity: 1..250=Low, 251..500=Medium, 501..750=High, 751..1000=Urgent
   Cfg_HiSeverity : ALIAS FOR Hi.Cfg_Severity;   // High Alarm Severity: 1..250=Low, 251..500=Medium, 501..750=High, 751..1000=Urgent
   Cfg_LoSeverity : ALIAS FOR Lo.Cfg_Severity;   // Low Alarm Severity: 1..250=Low, 251..500=Medium, 501..750=High, 751..1000=Urgent
   Cfg_LoLoSeverity : ALIAS FOR LoLo.Cfg_Severity;   // Low-Low Alarm Severity: 1..250=Low, 251..500=Medium, 501..750=High, 751..1000=Urgent
   Cfg_FailSeverity : ALIAS FOR Fail.Cfg_Severity;   // Failure Alarm Severity: 1..250=Low, 251..500=Medium, 501..750=High, 751..1000=Urgent
   Cfg_InpRawMin : REAL;   // Input (unscaled) Minimum for Scaling
   Cfg_InpRawMax : REAL := 100.0;   // Input (unscaled) Maximum for Scaling
   Cfg_PVEUMin : REAL;   // PV (Output) Minimum for Scaling to EU
   Cfg_PVEUMax : REAL := 100.0;   // PV (Output) Maximum for Scaling to EU
   Cfg_FiltTC : REAL;   // PV Filter Time Constant (s), 0.0 = unfiltered
   Cfg_HiHiDB : REAL := 1.0;   // High-High Status Deadband (EU)
   Cfg_HiHiOnDly : ALIAS FOR HiHiGate.Cfg_OnDly;   // Minimum time above High-High Limit to raise Status (s)
   Cfg_HiHiOffDly : ALIAS FOR HiHiGate.Cfg_OffDly;   // Minimum time below High-High Limit (minus deadband) to clear Status (s)
   Cfg_HiHiGateDly : ALIAS FOR HiHiGate.Cfg_GateDly;   // High-High Status Gate Delay (s)
   Cfg_HiDB : REAL := 1.0;   // High Status Deadband (EU)
   Cfg_HiOnDly : ALIAS FOR HiGate.Cfg_OnDly;   // Minimum time above High Limit to raise Status (s)
   Cfg_HiOffDly : ALIAS FOR HiGate.Cfg_OffDly;   // Minimum time below High Limit (minus deadband) to clear Status (s)
   Cfg_HiGateDly : ALIAS FOR HiGate.Cfg_GateDly;   // High Status Gate Delay (s)
   Cfg_LoDB : REAL := 1.0;   // Low Status Deadband (EU)
   Cfg_LoOnDly : ALIAS FOR LoGate.Cfg_OnDly;   // Minimum time below Low Limit to raise Status (s)
   Cfg_LoOffDly : ALIAS FOR LoGate.Cfg_OffDly;   // Minimum time above Low Limit (plus deadband) to clear Status (s)
   Cfg_LoGateDly : ALIAS FOR LoGate.Cfg_GateDly;   // Low Status Gate Delay (s)
   Cfg_LoLoDB : REAL := 1.0;   // Low-Low Status Deadband (EU)
   Cfg_LoLoOnDly : ALIAS FOR LoLoGate.Cfg_OnDly;   // Minimum time below Low-Low Limit to raise Status (s)
   Cfg_LoLoOffDly : ALIAS FOR LoLoGate.Cfg_OffDly;   // Minimum time above Low-Low Limit (plus deadband) to clear Status (s)
   Cfg_LoLoGateDly : ALIAS FOR LoLoGate.Cfg_GateDly;   // Low-Low Status Gate Delay (s)
   Cfg_FailHiLim : REAL := 103.958336;   // Out-of-Range (fail) High Limit (EU)
   Cfg_FailLoLim : REAL := -2.0833333;   // Out-of-Range (fail) Low Limit (EU)
   Cfg_FailDB : REAL := 0.41666666;   // Out-of-Range (fail) High/Low Deadband (EU)
   Cfg_FailOnDly : ALIAS FOR FailGate.Cfg_OnDly;   // Minimum time Bad or Out of Range to raise Fail Status (s)
   Cfg_FailOffDly : ALIAS FOR FailGate.Cfg_OffDly;   // Minimum time OK or In Range to clear Fail Status (s)
   Cfg_FailGateDly : ALIAS FOR FailGate.Cfg_GateDly;   // Fail Status Gate Delay (s)
   PSet_Owner : DINT;   // Program Owner Request ID (non-zero) or Release (zero)
   PSet_HiHiLim : REAL := 1.5e+38;   // Program-Entered High-High Status Threshold (EU)
   PSet_HiLim : REAL := 1.5e+38;   // Program-Entered High Status Threshold (EU)
   PSet_LoLim : REAL := -1.5e+38;   // Program-Entered Low Status Threshold (EU)
   PSet_LoLoLim : REAL := -1.5e+38;   // Program-Entered Low-Low Status Threshold (EU)
   MSet_SubstPV : REAL;   // Maintenance-Entered Substitute PV (EU)
   OSet_HiHiLim : REAL := 1.5e+38;   // Operator-Entered High-High Status Threshold (EU)
   OSet_HiLim : REAL := 1.5e+38;   // Operator-Entered High Status Threshold (EU)
   OSet_LoLim : REAL := -1.5e+38;   // Operator-Entered Low Status Threshold (EU)
   OSet_LoLoLim : REAL := -1.5e+38;   // Operator-Entered Low-Low Status Threshold (EU)
   Set_SimPV : REAL;   // PV used in Simulation (Inp_Sim=1) (EU)
   PCmd_ClearCapt : BOOL;   // Program Command to Clear the captured min / max PV excursion values
   PCmd_Acq : ALIAS FOR Mode.PCmd_Acq;
   PCmd_Rel : ALIAS FOR Mode.PCmd_Rel;
   PCmd_Lock : ALIAS FOR Mode.PCmd_Lock;
   PCmd_Unlock : ALIAS FOR Mode.PCmd_Unlock;
   PCmd_Reset : BOOL;   // Program Command to Reset all Alarms requiring Reset
   PCmd_HiHiAck : ALIAS FOR HiHi.PCmd_Ack;   // Program Command to Acknowledge High-High Alarm
   PCmd_HiHiSuppress : ALIAS FOR HiHi.PCmd_Suppress;   // Program Command to Suppress High-High Alarm
   PCmd_HiHiUnsuppress : ALIAS FOR HiHi.PCmd_Unsuppress;   // Program Command to Unsuppress High-High Alarm
   PCmd_HiHiUnshelve : ALIAS FOR HiHi.PCmd_Unshelve;   // Program Command to Unshelve High-High Alarm
   PCmd_HiAck : ALIAS FOR Hi.PCmd_Ack;   // Program Command to Acknowledge High Alarm
   PCmd_HiSuppress : ALIAS FOR Hi.PCmd_Suppress;   // Program Command to Suppress High Alarm
   PCmd_HiUnsuppress : ALIAS FOR Hi.PCmd_Unsuppress;   // Program Command to Unsuppress High Alarm
   PCmd_HiUnshelve : ALIAS FOR Hi.PCmd_Unshelve;   // Program Command to Unshelve High Alarm
   PCmd_LoAck : ALIAS FOR Lo.PCmd_Ack;   // Program Command to Acknowledge Low Alarm
   PCmd_LoSuppress : ALIAS FOR Lo.PCmd_Suppress;   // Program Command to Suppress Low Alarm
   PCmd_LoUnsuppress : ALIAS FOR Lo.PCmd_Unsuppress;   // Program Command to Unsuppress Low Alarm
   PCmd_LoUnshelve : ALIAS FOR Lo.PCmd_Unshelve;   // Program Command to Unshelve Low Alarm
   PCmd_LoLoAck : ALIAS FOR LoLo.PCmd_Ack;   // Program Command to Acknowledge Low-Low Alarm
   PCmd_LoLoSuppress : ALIAS FOR LoLo.PCmd_Suppress;   // Program Command to Suppress Low-Low Alarm
   PCmd_LoLoUnsuppress : ALIAS FOR LoLo.PCmd_Unsuppress;   // Program Command to Unsuppress Low-Low Alarm
   PCmd_LoLoUnshelve : ALIAS FOR LoLo.PCmd_Unshelve;   // Program Command to Unshelve Low-Low Alarm
   PCmd_FailAck : ALIAS FOR Fail.PCmd_Ack;   // Program Command to Acknowldege Analog Input Failure Alarm
   PCmd_FailSuppress : ALIAS FOR Fail.PCmd_Suppress;   // Program Command to Suppress Analog Input Failure Alarm
   PCmd_FailUnsuppress : ALIAS FOR Fail.PCmd_Unsuppress;   // Program Command to Unsuppress Analog Input Failure Alarm
   PCmd_FailUnshelve : ALIAS FOR Fail.PCmd_Unshelve;   // Program Command to Unshelve Analog Input Failure Alarm
   MCmd_SubstPV : BOOL;   // Maintenance Command to use Substitute PV (override input)
   MCmd_InpPV : BOOL;   // Maintenance Command to use Input PV (normal)
   OCmd_ClearCapt : BOOL;   // Operator Command to Clear the captured min / max PV excursion values
   MCmd_Acq : ALIAS FOR Mode.MCmd_Acq;
   MCmd_Rel : ALIAS FOR Mode.MCmd_Rel;
   OCmd_AcqLock : ALIAS FOR Mode.OCmd_AcqLock;
   OCmd_Unlock : ALIAS FOR Mode.OCmd_UnlockRel;
   OCmd_Reset : BOOL;   // Operator Command to Reset all Alarms requiring Reset
   OCmd_ResetAckAll : BOOL;   // Operator Command to Reset and Acknowledge all Alarms
END_VAR
VAR_OUTPUT
   Val : REAL; {access Read Only, visible}   // Analog Value (after Substitute PV, if used)
   Val_InpPV : REAL; {access Read Only, visible}   // Analog Input Value (actual, before Substitute PV selection)
   Val_PVMinCapt : REAL := 1.5e+38; {access Read Only}   // Captured PV Minimum (excursion) since last cleared
   Val_PVMaxCapt : REAL := -1.5e+38; {access Read Only}   // Captured PV Maximum (excursion) since last cleared
   Val_PVEUMin : REAL; {access Read Only}   // Minimum of scaled range = MIN (Cfg_PVEUMin, Cfg_PVEUMax)
   Val_PVEUMax : REAL := 100.0; {access Read Only}   // Maximum of scaled range = MAX (Cfg_PVEUMin, Cfg_PVEUMax)
   SrcQ_IO : DINT; {access Read Only}   // Source and Quality of primary I/O (enumeration)
   SrcQ : DINT; {access Read Only}   // Source and Quality of primary Val/Sts (enumeration)
   Val_Fault : DINT; {access Read Only}   // Device Fault Status 0=none, 20=Lo, 21=Hi, 24=LoLo, 25=HiHi, 32=Fail, 34=CfgErr
   Val_Mode : ALIAS FOR Mode.Val; {access Read Only}
   Val_Owner : DINT; {access Read Only}   // Current Object Owner ID (0=not owned)
   Val_Notify : DINT; {access Read Only}   // Current Alarm Level and Acknowledgement (enumeration)
   Val_HiHiLim : REAL := 1.5e+38; {access Read Only, visible}   // Current High-High Status Threshold
   Val_HiLim : REAL := 1.5e+38; {access Read Only, visible}   // Current High Status Threshold
   Val_LoLim : REAL := -1.5e+38; {access Read Only, visible}   // Current Low Status Threshold
   Val_LoLoLim : REAL := -1.5e+38; {access Read Only, visible}   // Current Low-Low Status Threshold
   Sts_SubstPV : BOOL; {access Read Only}   // 1=Using Substitute PV (Input being overridden)
   Sts_InpPV : BOOL := 1; {access Read Only}   // 1=Using Input PV (normal)
   Sts_PVBad : BOOL; {access Read Only}   // 1=PV Bad quality or Out of Range
   Sts_PVUncertain : BOOL; {access Read Only}   // 1=PV Value is Uncertain (quality)
   Sts_MaintByp : BOOL; {access Read Only}   // 1=A Maintenance Bypass is Active, display icon
   Sts_AlmInh : BOOL; {access Read Only}   // 1=An Alarm is Shelved, Disabled or Suppressed: display icon
   Sts_Err : BOOL; {access Read Only, visible}   // 1=Error in Config (see detail Err_ bits for reason), display icon
   Err_Raw : BOOL; {access Read Only}   // 1=Error in Config: Raw Input Scaling Min = Max
   Err_EU : BOOL; {access Read Only}   // 1=Error in Config: Scaled EU Min = Max
   Err_Timer : BOOL; {access Read Only}   // 1=Error in Config: On Delay, Off Delay, Gate Delay Time Invalid (use 0 to 2147483 s)
   Err_Filt : BOOL; {access Read Only}   // 1=Error in Config: PV filter params (RateTime, TC)
   Err_DB : BOOL; {access Read Only}   // 1=Error in Config: a Status Deadband is < 0.0
   Err_Alarm : BOOL; {access Read Only}   // 1=Error in Config: Alarm Min On Time, Shelf Time, Severity
   Sts_Maint : ALIAS FOR Mode.Sts_Maint; {access Read Only}
   Sts_Prog : ALIAS FOR Mode.Sts_Prog; {access Read Only}
   Sts_Oper : ALIAS FOR Mode.Sts_Oper; {access Read Only}
   Sts_ProgOperLock : ALIAS FOR Mode.Sts_ProgOperLock; {access Read Only}
   Sts_NoMode : ALIAS FOR Mode.Sts_NoMode; {access Read Only}
   Sts_MAcqRcvd : ALIAS FOR Mode.Sts_MAcqRcvd; {access Read Only}
   Sts_HiHiCmp : ALIAS FOR HiHiGate.Inp;   // PV High-High comparison result 1=High-High
   Sts_HiHiGate : ALIAS FOR HiHiGate.Sts_Gate; {access Read Only}   // PV High-High Gate Delay Status, 1=done
   Sts_HiHi : ALIAS FOR HiHi.Inp;   // 1=Analog Input is above High-High limit
   Alm_HiHi : ALIAS FOR HiHi.Alm;   // 1=Analog Input is in High-High Alarm
   Ack_HiHi : ALIAS FOR HiHi.Ack;   // 1=High-High Alarm has been acknowledged
   Sts_HiHiDisabled : ALIAS FOR HiHi.Disabled;   // 1=High-High Alarm has been Disabled by Maintenancy
   Sts_HiHiSuppressed : ALIAS FOR HiHi.Suppressed;   // 1=High-High Alarm has been Suppressed by Program
   Sts_HiHiShelved : ALIAS FOR HiHi.Shelved;   // 1=High-High Alarm has been Shelved by Operator
   Sts_HiCmp : ALIAS FOR HiGate.Inp;   // PV High comparison result 1=High
   Sts_HiGate : ALIAS FOR HiGate.Sts_Gate; {access Read Only}   // PV High Gate Delay Status, 1=done
   Sts_Hi : ALIAS FOR Hi.Inp;   // 1=Analog Input is above High limit
   Alm_Hi : ALIAS FOR Hi.Alm;   // 1=Analog Input is in High Alarm
   Ack_Hi : ALIAS FOR Hi.Ack;   // 1=High Alarm has been acknowledged
   Sts_HiDisabled : ALIAS FOR Hi.Disabled;   // 1=High Alarm has been Disabled by Maintenance
   Sts_HiSuppressed : ALIAS FOR Hi.Suppressed;   // 1=High Alarm has been Suppressed by Program
   Sts_HiShelved : ALIAS FOR Hi.Shelved;   // 1=High Alarm has been Shelved by Operator
   Sts_LoCmp : ALIAS FOR LoGate.Inp;   // PV Low comparison result 1=Low
   Sts_LoGate : ALIAS FOR LoGate.Sts_Gate; {access Read Only}   // PV Low Gate Delay Status, 1=done
   Sts_Lo : ALIAS FOR Lo.Inp;   // 1=Analog Input is below Low limit
   Alm_Lo : ALIAS FOR Lo.Alm;   // 1=Analog Input is in Low Alarm
   Ack_Lo : ALIAS FOR Lo.Ack;   // 1=Low Alarm has been acknowledged
   Sts_LoDisabled : ALIAS FOR Lo.Disabled;   // 1=Low Alarm has been Disabled by Maintenance
   Sts_LoSuppressed : ALIAS FOR Lo.Suppressed;   // 1=Low Alarm has been Suppressed by Program
   Sts_LoShelved : ALIAS FOR Lo.Shelved;   // 1=Low Alarm has been Shelved by Operator
   Sts_LoLoCmp : ALIAS FOR LoLoGate.Inp;   // PV Low-Low comparison result 1=Low-Low
   Sts_LoLoGate : ALIAS FOR LoLoGate.Sts_Gate; {access Read Only}   // PV Low-Low Gate Delay Status, 1=done
   Sts_LoLo : ALIAS FOR LoLo.Inp;   // 1=Analog Input is below Low-Low limit
   Alm_LoLo : ALIAS FOR LoLo.Alm;   // 1=Analog Input is in Low-Low Alarm
   Ack_LoLo : ALIAS FOR LoLo.Ack;   // 1=Low-Low Alarm has been acknowledged
   Sts_LoLoDisabled : ALIAS FOR LoLo.Disabled;   // 1=Low-Low Alarm has been Disabled by Maintenance
   Sts_LoLoSuppressed : ALIAS FOR LoLo.Suppressed;   // 1=Low-Low Alarm has been Suppressed by Program
   Sts_LoLoShelved : ALIAS FOR LoLo.Shelved;   // 1=Low-Low Alarm has been Shelved by Operator
   Sts_FailCmp : ALIAS FOR FailGate.Inp;   // PV Fail comparison result 1=Out of Range
   Sts_FailGate : ALIAS FOR FailGate.Sts_Gate; {access Read Only}   // PV Fail Gate Delay Status, 1=done
   Sts_Fail : ALIAS FOR Fail.Inp;   // 1=Analog Input is Out of Range or PV Bad
   Alm_Fail : ALIAS FOR Fail.Alm;   // 1=Analog Input Failure Alarm (PV Bad or Out of Range)
   Ack_Fail : ALIAS FOR Fail.Ack;   // 1=Analog Input Failure Alarm has been acknowledged
   Sts_FailDisabled : ALIAS FOR Fail.Disabled;   // 1=Analog input Failure Alarm has been Disabled by Maintenance
   Sts_FailSuppressed : ALIAS FOR Fail.Suppressed;   // 1=Analog Input Failure Alarm has been Suppressed by Program
   Sts_FailShelved : ALIAS FOR Fail.Shelved;   // 1=Analog Input Failure Alarm has been Shelved by Operator
   Rdy_SubstPV : BOOL; {access Read Only}   // 1=Ready for MCmd_SubstPV
   Rdy_InpPV : BOOL; {access Read Only}   // 1=Ready for MCmd_InpPV
   Rdy_Reset : BOOL; {access Read Only}   // 1=At least one Alarm requires Reset
   Rdy_ResetAckAll : BOOL; {access Read Only}   // 1=At least one Alarm requires Reset or Acknowledgement
   Rdy_OSet : BOOL; {access Read Only}   // 1=Ready to receive OSets (enables data entry fields)
   P_AIn : BOOL;   // Unique Parameter Name for auto - discovery
END_VAR
VAR
   LoLo : P_Alarm := (Cfg_AckReqd := 1, Cfg_AllowShelve := 1, Cfg_AllowDisable := 1, Cfg_PCmdClear := 1, Cfg_Severity := 750, Cfg_AlmMinOnT := 5, PCfg_AllowExist := 1, Ack := 1);   // Low-Low Alarm
   Lo : P_Alarm := (Cfg_AckReqd := 1, Cfg_AllowShelve := 1, Cfg_AllowDisable := 1, Cfg_PCmdClear := 1, Cfg_Severity := 500, Cfg_AlmMinOnT := 5, PCfg_AllowExist := 1, Ack := 1);   // Low Alarm
   Hi : P_Alarm := (Cfg_AckReqd := 1, Cfg_AllowShelve := 1, Cfg_AllowDisable := 1, Cfg_PCmdClear := 1, Cfg_Severity := 500, Cfg_AlmMinOnT := 5, PCfg_AllowExist := 1, Ack := 1);   // High Alarm
   HiHi : P_Alarm := (Cfg_AckReqd := 1, Cfg_AllowShelve := 1, Cfg_AllowDisable := 1, Cfg_PCmdClear := 1, Cfg_Severity := 750, Cfg_AlmMinOnT := 5, PCfg_AllowExist := 1, Ack := 1);   // High-High Alarm
   Mode : P_Mode := (Cfg_PCmdClear := 1, Cfg_OvrdOverLock := 1, Sts_Oper := 1, Rdy_MRel := 1, Rdy_OAcq := 1);   // Analog Input Mode Selection
   Cfg_EU : String_4 := '%';   // Engineering Units for display on HMI
   Cfg_Tag : STRING_12;   // Tagname for display on HMI
   Cfg_Label : STRING_12;   // Label for graphic symbol displayed on HMI
   Cfg_Desc : STRING_20;   // Description for display on HMI
   Fail : P_Alarm := (Cfg_AckReqd := 1, Cfg_AllowShelve := 1, Cfg_AllowDisable := 1, Cfg_PCmdClear := 1, Cfg_Severity := 1000, Cfg_AlmMinOnT := 5, PCfg_AllowExist := 1, Ack := 1);   // Analog Input Failure Alarm (bad quality or out of range)
   Wrk_Notify : DINT; {access None}   // Buffer for building Val_Notify
   Inf_Tab : DINT;   // Tab to display (FTView ME)
   Wrk_SrcQ : DINT; {access None}   // Register for building Source / Quality enumeration
   Wrk_Fault : DINT; {access None}   // Buffer for building Val_Fault
   Wrk_SubstPV : BOOL; {access None}   // Internal flag: Using Substitute PV
   Wrk_UnfiltPV : REAL; {access None}   // Unfiltered PV, input to 1st order filter
   Wrk_Alpha : REAL; {access None}   // Filter multiplier = (1 / (1+TC/dT) )
   Wrk_ScanT : TIMER := (PRE := 2147483647); {access None}   // Scan Timer (milliseconds, always runs)
   Wrk_ScanTime : REAL; {access None}   // Time since this instance was last scanned
   Wrk_FiltPV : REAL; {access None}   // Filtered PV
   Wrk_ValidONS : BOOL; {access None}   // Selected PV goes from Infinite or Not a Number to VALID
   Wrk_SelPVDINT : DINT; {access None}   // Selected PV check for Infinite or Non A Number
   Wrk_SelPVInfNaN : BOOL; {access None}   // Selected PV (Input or Substitute) is Infinite or NaN
   Wrk_Fail : BOOL; {access None}   // Internal flag: Fail Status
   Wrk_LoLo : BOOL; {access None}   // Internal flag: Low-Low Status
   Wrk_Lo : BOOL; {access None}   // Internal flag: Low Status
   Wrk_Hi : BOOL; {access None}   // Internal flag: High Status
   Wrk_HiHi : BOOL; {access None}   // Internal flag: High-High Status
   FailGate : P_Gate := (Inp_Gate := 1);   // Fail Alarm Gate / Delay Block
   LoLoGate : P_Gate := (Inp_Gate := 1);   // Low-Low Alarm Gate / Delay Block
   LoGate : P_Gate := (Inp_Gate := 1);   // Low Alarm Gate / Delay Block
   HiHiGate : P_Gate := (Inp_Gate := 1);   // High-High Alarm Gate / Delay Block
   HiGate : P_Gate := (Inp_Gate := 1);   // High Alarm Gate / Delay Block
   Wrk_InpInfNaN : BOOL; {access None}   // Input is Infinite or Not a Number
   Wrk_InpDINT : DINT; {access None}   // Input REAL bit pattern as a DINT (check for Inf/NaN)
   Wrk_InpFail : BOOL; {access None}   // Input Fail: out of range
END_VAR

ROUTINE EnableInFalse   (* ladder *)
// Off-Scan: no Val update or alarm checking.  PV Bad Quality ("stale") is asserted.
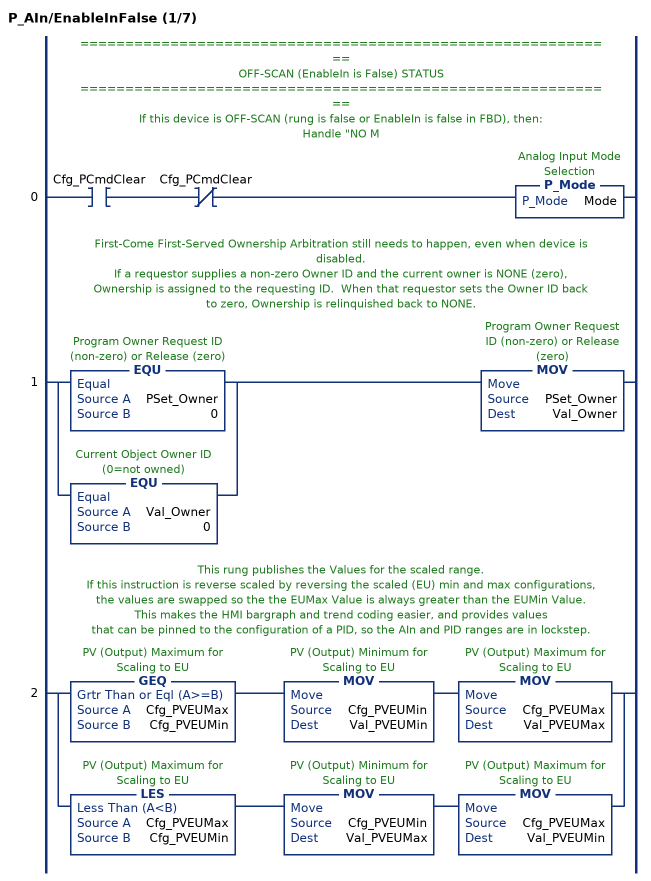
   // ============================================================
   // OFF-SCAN (EnableIn is False) STATUS
   // ============================================================
   // If this device is OFF-SCAN (rung is false or EnableIn is false in FBD), then:
   // Handle "NO M
   0: XIC(Cfg_PCmdClear)XIO(Cfg_PCmdClear)P_Mode(Mode);
   // First-Come First-Served Ownership Arbitration still needs to happen, even when device is disabled.
   // If a requestor supplies a non-zero Owner ID and the current owner is NONE (zero),
   // Ownership is assigned to the requesting ID.  When that requestor sets the Owner ID back
   // to zero, Ownership is relinquished back to NONE.
   1: [EQU(PSet_Owner,0) ,EQU(Val_Owner,0) ]MOV(PSet_Owner,Val_Owner);
   // This rung publishes the Values for the scaled range.
   // If this instruction is reverse scaled by reversing the scaled (EU) min and max configurations,
   // the values are swapped so the the EUMax Value is always greater than the EUMin Value.
   // This makes the HMI bargraph and trend coding easier, and provides values
   // that can be pinned to the configuration of a PID, so the AIn and PID ranges are in lockstep.
   2: [GEQ(Cfg_PVEUMax,Cfg_PVEUMin) MOV(Cfg_PVEUMin,Val_PVEUMin) MOV(Cfg_PVEUMax,Val_PVEUMax) ,LES(Cfg_PVEUMax,Cfg_PVEUMin) MOV(Cfg_PVEUMin,Val_PVEUMax) MOV(Cfg_PVEUMax,Val_PVEUMin) ];
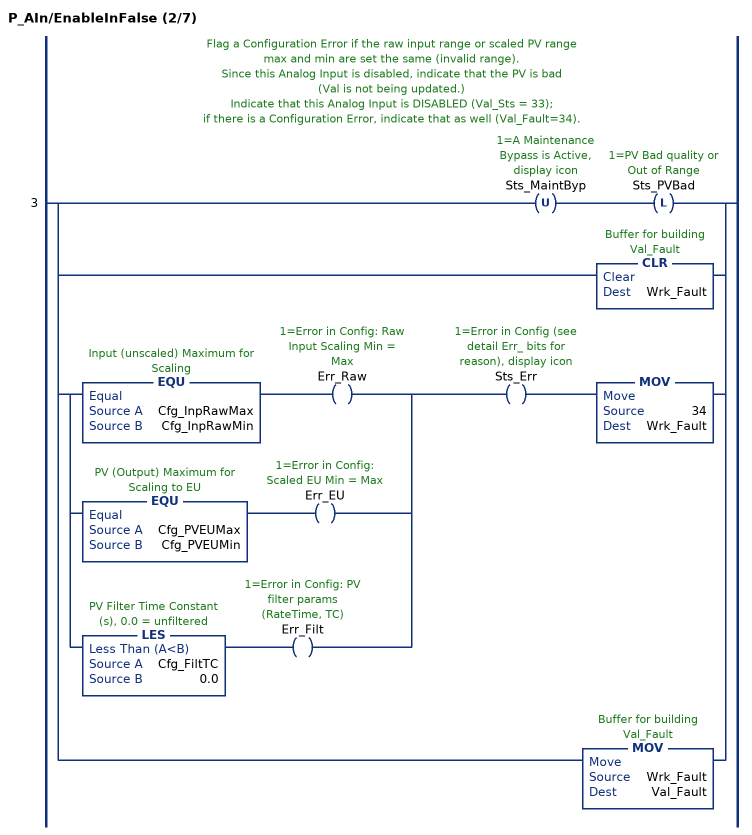
   // Flag a Configuration Error if the raw input range or scaled PV range
   // max and min are set the same (invalid range).
   // Since this Analog Input is disabled, indicate that the PV is bad
   // (Val is not being updated.)
   // Indicate that this Analog Input is DISABLED (Val_Sts = 33);
   // if there is a Configuration Error, indicate that as well (Val_Fault=34).
   3: [OTU(Sts_MaintByp) OTL(Sts_PVBad) ,CLR(Wrk_Fault) ,[EQU(Cfg_InpRawMax,Cfg_InpRawMin) OTE(Err_Raw) ,EQU(Cfg_PVEUMax,Cfg_PVEUMin) OTE(Err_EU) ,LES(Cfg_FiltTC,0.0) OTE(Err_Filt) ] OTE(Sts_Err) MOV(34,Wrk_Fault) ,MOV(Wrk_Fault,Val_Fault) ];
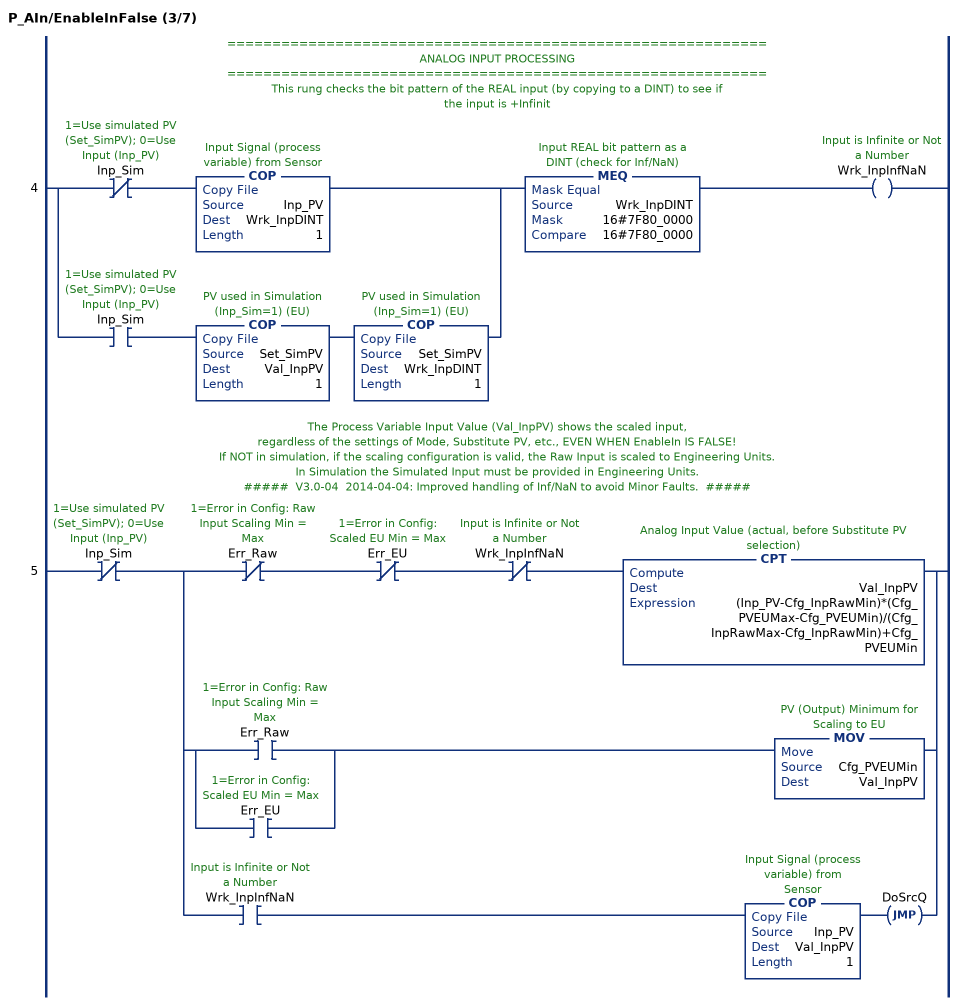
   // ============================================================
   // ANALOG INPUT PROCESSING
   // ============================================================
   // This rung checks the bit pattern of the REAL input (by copying to a DINT) to see if
   // the input is +Infinit
   4: [XIO(Inp_Sim) COP(Inp_PV,Wrk_InpDINT,1) ,XIC(Inp_Sim) COP(Set_SimPV,Val_InpPV,1) COP(Set_SimPV,Wrk_InpDINT,1) ]MEQ(Wrk_InpDINT,16#7F80_0000,16#7F80_0000)OTE(Wrk_InpInfNaN);
   // The Process Variable Input Value (Val_InpPV) shows the scaled input,
   // regardless of the settings of Mode, Substitute PV, etc., EVEN WHEN EnableIn IS FALSE!
   // If NOT in simulation, if the scaling configuration is valid, the Raw Input is scaled to Engineering Units.
   // In Simulation the Simulated Input must be provided in Engineering Units.
   // #####  V3.0-04  2014-04-04: Improved handling of Inf/NaN to avoid Minor Faults.  #####
   5: XIO(Inp_Sim)[XIO(Err_Raw) XIO(Err_EU) XIO(Wrk_InpInfNaN) CPT(Val_InpPV,(Inp_PV-Cfg_InpRawMin)*(Cfg_PVEUMax-Cfg_PVEUMin)/(Cfg_InpRawMax-Cfg_InpRawMin)+Cfg_PVEUMin) ,[XIC(Err_Raw) ,XIC(Err_EU) ] MOV(Cfg_PVEUMin,Val_InpPV) ,XIC(Wrk_InpInfNaN) COP(Inp_PV,Val_InpPV,1) JMP(DoSrcQ) ];
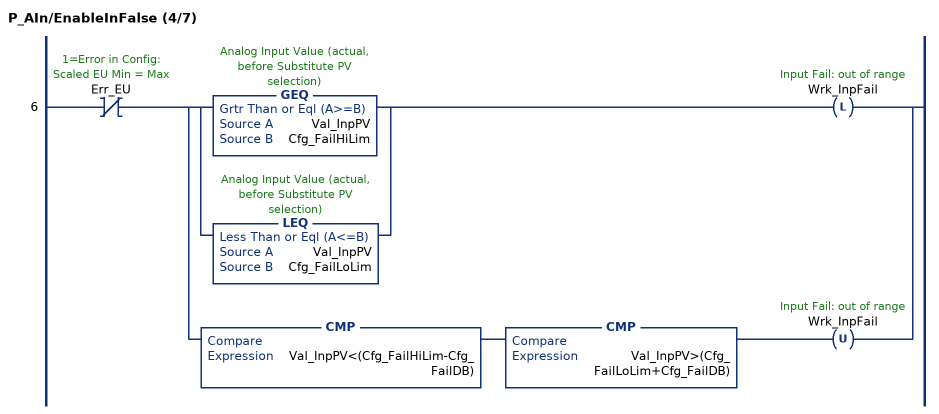
   6: XIO(Err_EU)[[GEQ(Val_InpPV,Cfg_FailHiLim) ,LEQ(Val_InpPV,Cfg_FailLoLim) ] OTL(Wrk_InpFail) ,CMP(Val_InpPV<(Cfg_FailHiLim-Cfg_FailDB)) CMP(Val_InpPV>(Cfg_FailLoLim+Cfg_FailDB)) OTU(Wrk_InpFail) ];
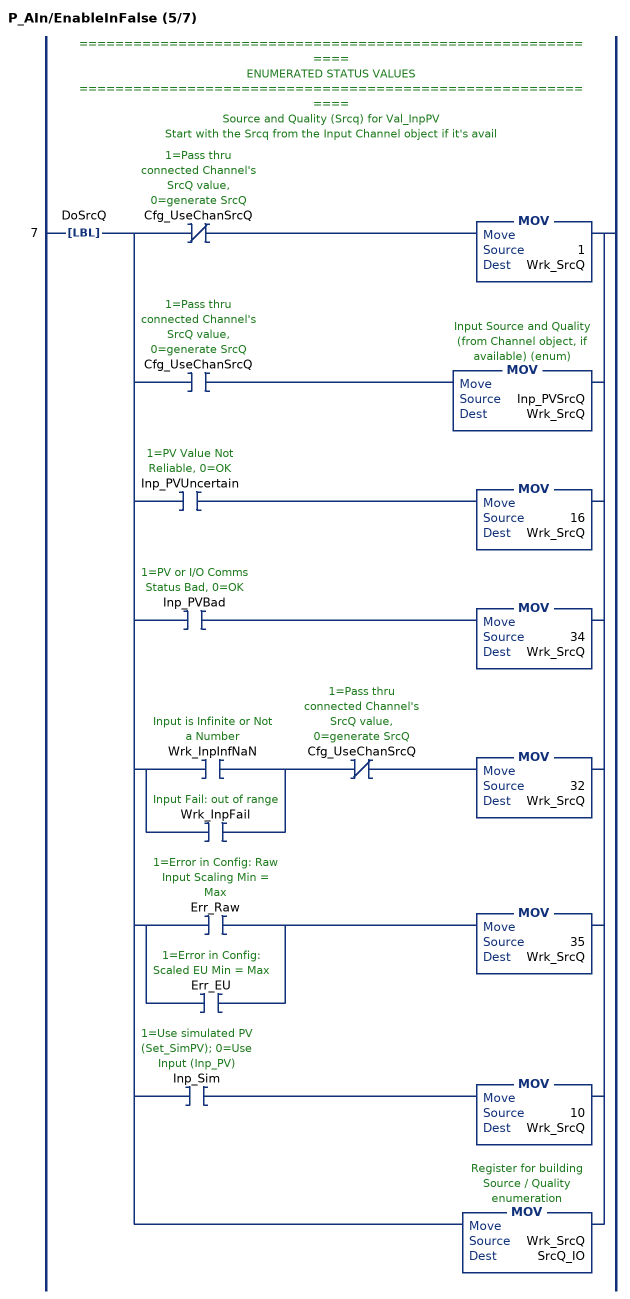
   // ============================================================
   // ENUMERATED STATUS VALUES
   // ============================================================
   // Source and Quality (Srcq) for Val_InpPV
   // Start with the Srcq from the Input Channel object if it's avail
   7: LBL(DoSrcQ)[XIO(Cfg_UseChanSrcQ) MOV(1,Wrk_SrcQ) ,XIC(Cfg_UseChanSrcQ) MOV(Inp_PVSrcQ,Wrk_SrcQ) ,XIC(Inp_PVUncertain) MOV(16,Wrk_SrcQ) ,XIC(Inp_PVBad) MOV(34,Wrk_SrcQ) ,[XIC(Wrk_InpInfNaN) ,XIC(Wrk_InpFail) ] XIO(Cfg_UseChanSrcQ) MOV(32,Wrk_SrcQ) ,[XIC(Err_Raw) ,XIC(Err_EU) ] MOV(35,Wrk_SrcQ) ,XIC(Inp_Sim) MOV(10,Wrk_SrcQ) ,MOV(Wrk_SrcQ,SrcQ_IO) ];
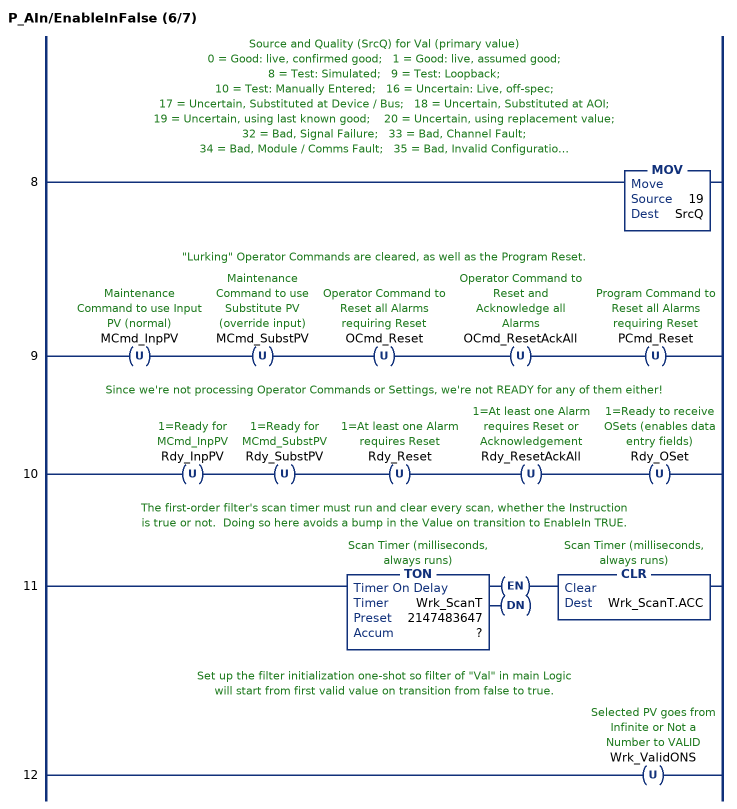
   // Source and Quality (SrcQ) for Val (primary value)
   // 0 = Good: live, confirmed good;   1 = Good: live, assumed good;
   // 8 = Test: Simulated;   9 = Test: Loopback;
   // 10 = Test: Manually Entered;   16 = Uncertain: Live, off-spec;
   // 17 = Uncertain, Substituted at Device / Bus;   18 = Uncertain, Substituted at AOI;
   // 19 = Uncertain, using last known good;    20 = Uncertain, using replacement value;
   // 32 = Bad, Signal Failure;   33 = Bad, Channel Fault;
   // 34 = Bad, Module / Comms Fault;   35 = Bad, Invalid Configuration
   // #####  V3.1-00  2014-06-30:  Added rung for Source/Quality enumerations.  #####
   8: MOV(19,SrcQ);
   // "Lurking" Operator Commands are cleared, as well as the Program Reset.
   9: OTU(MCmd_InpPV)OTU(MCmd_SubstPV)OTU(OCmd_Reset)OTU(OCmd_ResetAckAll)OTU(PCmd_Reset);
   // Since we're not processing Operator Commands or Settings, we're not READY for any of them either!
   10: OTU(Rdy_InpPV)OTU(Rdy_SubstPV)OTU(Rdy_Reset)OTU(Rdy_ResetAckAll)OTU(Rdy_OSet);
   // The first-order filter's scan timer must run and clear every scan, whether the Instruction
   // is true or not.  Doing so here avoids a bump in the Value on transition to EnableIn TRUE.
   11: TON(Wrk_ScanT,?,?)CLR(Wrk_ScanT.ACC);
   // Set up the filter initialization one-shot so filter of "Val" in main Logic
   // will start from first valid value on transition from false to true.
   12: OTU(Wrk_ValidONS);
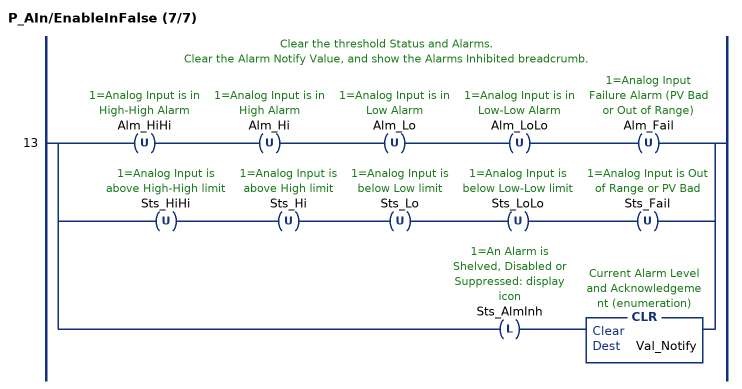
   // Clear the threshold Status and Alarms.
   // Clear the Alarm Notify Value, and show the Alarms Inhibited breadcrumb.
   13: [OTU(Alm_HiHi) OTU(Alm_Hi) OTU(Alm_Lo) OTU(Alm_LoLo) OTU(Alm_Fail) ,OTU(Sts_HiHi) OTU(Sts_Hi) OTU(Sts_Lo) OTU(Sts_LoLo) OTU(Sts_Fail) ,OTL(Sts_AlmInh) CLR(Val_Notify) ];
END_ROUTINE
